(************************************************************************************)
(*							Beckhoff Automation Poland								*)
(*								FB_ShortLongTrig v2									*)
(*									2.04.2012										*)
(*	Bloczek do rozpoznania długiego/krotkiego wcisniecia przycisku- wyjscia			*)
(*__________________________________________________________________________________*)
FUNCTION_BLOCK FB_ShortLongTrig
VAR_INPUT
	bSwitch: 	BOOL; (*Przycisk*)
	tLong: 		TIME; (*Czas dlugiego wcisniecia*)
END_VAR
VAR_OUTPUT
	bShort: 	BOOL; (*TRUE gdy krotkie*)
	bLong: 		BOOL;(*TRUE gdy dlugie*)
END_VAR
VAR
	t1: 		TON;
	ft1: 		F_TRIG;
END_VAR

ft1(CLK:= bSwitch , Q=> );
IF ft1.Q THEN
	bLong := t1.Q;
	bShort := NOT t1.Q;
ELSE
	bLong := FALSE;
	bShort := FALSE;
END_IF
t1(IN:= bSwitch, PT:= tLong, Q=> , ET=> );

END_FUNCTION_BLOCK

(* stored: Version 1.1.0.1, ProductVersion 3.1.4020.3
   POU FB_ShortLongTrig: Id {eba27b1c-a1ee-41df-91a6-e378de26162a}, SpecialFunc None *)
